TYPE DUT_UpdatePartLocationsAndProcessingData :
STRUCT
	return_value	: DINT;
	Data	: STRING(DB.MAX_STRING_SIZE);
END_STRUCT
END_TYPE

(* stored: Version 1.1.0.1, ProductVersion 3.1.4024.15
   DUT DUT_UpdatePartLocationsAndProcessingData: Id {6fcdc8ee-c381-4e2b-9082-d746bb80b2be} *)
